Fanuc KAREL source: port_LAO.kl

PROGRAM TP
%NOLOCKGROUP
VAR
 x: INTEGER
BEGIN
 x = LAO[3]
END TP
